TYPE DigitalInputBase_50022E7B :
STRUCT
END_STRUCT
END_TYPE

(* stored: Version 1.2.0.0, ProductVersion 3.1.4024.9
   DUT DigitalInputBase_50022E7B: Id {f7830df3-6433-4635-8a67-39701336b704} *)
